// Brief: Master Arm Orientation Matching
FUNCTION_BLOCK PUBLIC FB_StateCtrlMatching EXTENDS FB_MasterArmCtrlBase
VAR_INPUT
END_VAR
VAR_OUTPUT
END_VAR
VAR
	// master-slave orientation match threshold
	m_matchAngleThres :LREAL := 2*g_deg2Rad;
	
	m_cmdRotInMonitor :Mat3d;
	
	m_initSolvedJntPos, m_iteSovlvedJntPos :Vec7d;
	m_IKSuccess :BOOL;
	
	m_matchTrajPlanner : FB_TrajMoveJ;
	m_targetJntPos :Vec7d;
	
	m_maxMatchJntVel:Vec7d:=[1.0, 1.0, 1.0, 2*pi, 3*pi, 3*pi, 5*pi];
	m_maxMatchJntAcc:Vec7d:=[1.0, 1.0, 1.0,  8*pi, 12*pi, 12*pi, 20*pi];
	m_maxMatchJntJerk:Vec7d:=[7(100.0)];
	
	m_rotErrAng :LREAL;

END_VAR

// override this function in each exact controller
METHOD PROTECTED calcCmdJntPos : BOOL

VAR_IN_OUT CONSTANT
	i_slaveIdx :INT;
	i_shoulderPose :ST_Frame;
	i_masterArm :FB_MasterArm;
	i_slaveStatus :ST_SlaveStatus;
END_VAR
var 
	i,j : INT;

	mq4,mq5,mq6,mq7:LREAL;
	q4,q5,q6,q7:LREAL;

	rotErr:Mat3d;
	wristRotInJnt3, wristRotInJnt4 :Mat3d;
	rot, invRot :Mat3d;
	cycleNum:INT;
	
	jnt4MoveRange:LREAL;
	jnt5Bias, jnt4MoveScale :LREAL;
	
	cmdJntErr:Vec7d;

END_VAR
IF m_IKSuccess THEN 
	// check if planner is ready
	IF  m_matchTrajPlanner.isGene = FALSE THEN
		RETURN;
	END_IF
	
	// traj plan
	calcCmdJntPos :=m_matchTrajPlanner.evaluate(m_timePeriod, jntPos=> m_cmdJntPos, jntVel=>m_cmdJntVel, jntAcc=> m_cmdJntAcc);
	
	vecSub(m_targetJntPos, m_cmdJntPos, cmdJntErr);
	
	matTranspose(i_masterArm.curCartPose.m_rot, invRot);
	matMultiply(invRot, m_cmdCartPose.m_rot, rotErr);
	rot2AngAxis(rotErr, angle=>m_rotErrAng,axis=>);
	m_isFinished := m_timePeriod > m_matchTrajPlanner.duration AND  norm(cmdJntErr)<g_jntCtrlAngTolHigh and abs(m_rotErrAng)<g_jntCtrlAngTolHigh;
	
	RETURN;
END_IF

// command rotation in monitor
m_cmdRotInMonitor := i_slaveStatus.m_curArmPose[i_slaveIdx].m_rot;

// command rotation in master arm base
matTranspose(i_shoulderPose.m_rot, invRot);
matMultiply(invRot, m_cmdRotInMonitor, m_cmdCartPose.m_rot);
m_cmdCartPose.m_pos:= i_masterArm.curCartPose.m_pos;

// calculate current orientation error
matTranspose(i_masterArm.curCartPose.m_rot, invRot);
matMultiply(invRot, m_cmdCartPose.m_rot, rotErr);
rot2AngAxis(rotErr, angle=>m_rotErrAng,axis=>);

// try IK with optimized posture
rot:=calcJnt3Rotation(m_cmdJntPos[1],m_cmdJntPos[2],m_cmdJntPos[3]);
matTranspose(rot, invRot);
matMultiply(invRot, m_cmdCartPose.m_rot, wristRotInJnt3);
IF 1=i_masterArm.armIdx THEN
	m_IKSuccess := leftWristOptIK(wristRotInJnt3,q4=>q4, q5=>q5, q6=>q6, q7=>q7);
ELSE
	m_IKSuccess := rightWristOptIK(wristRotInJnt3,q4=>q4, q5=>q5, q6=>q6, q7=>q7);
END_IF

// try IK with joint4 at minimal limit
IF NOT m_IKSuccess THEN
	q4:= GVL_ArmJointParameters.g_minJntPos[i_masterArm.armIdx,4];
	
	rot:=calcJnt4Rotation(m_cmdJntPos[1],m_cmdJntPos[2],m_cmdJntPos[3],q4);
	matTranspose(rot, invRot);
	matMultiply(invRot, m_cmdCartPose.m_rot, wristRotInJnt4);
	m_IKSuccess := wristIK(wristRotInJnt4,i_masterArm, q5=>q5, q6=>q6, q7=>q7);
END_IF

// try IK with joint4 at maximum limit
IF NOT m_IKSuccess THEN
	q4:= GVL_ArmJointParameters.g_maxJntPos[i_masterArm.armIdx,4];
	
	rot:=calcJnt4Rotation(m_cmdJntPos[1],m_cmdJntPos[2],m_cmdJntPos[3],q4);
	matTranspose(rot, invRot);
	matMultiply(invRot, m_cmdCartPose.m_rot, wristRotInJnt4);
	m_IKSuccess := wristIK(wristRotInJnt4,i_masterArm, q5=>q5, q6=>q6, q7=>q7);
END_IF

// minimize joint4 move angle
IF m_IKSuccess THEN
	
	// minimize based on join5 posture
	jnt4MoveRange :=  i_masterArm.jnt4LinkToMotor(m_targetJntPos[2],m_targetJntPos[3],q4)-i_masterArm.curJntPos[4];
	jnt5Bias :=  LIMIT (0, ABS(q5-pi), pi/2);
	jnt4MoveRange := jnt4MoveRange * ABS(COS(jnt5Bias));
	
	// minimize based on cartesian error
	IF ABS(m_rotErrAng)< 5.0 * g_deg2Rad THEN
		jnt4MoveRange := 0.0;
	END_IF
	
	mq4:=  i_masterArm.jnt4MotorToLink(m_targetJntPos[2],m_targetJntPos[3],i_masterArm.curJntPos[4] + jnt4MoveRange) ;
	
	rot:=calcJnt4Rotation(m_cmdJntPos[1],m_cmdJntPos[2],m_cmdJntPos[3],mq4);
	matTranspose(rot, invRot);
	matMultiply(invRot, m_cmdCartPose.m_rot, wristRotInJnt4);
	IF wristIK(wristRotInJnt4,i_masterArm, q5=>mq5, q6=>mq6, q7=>mq7) THEN
		q4:=mq4;
		q5:=mq5;
		q6:=mq6;
		q7:=mq7;
	END_IF
END_IF

// traj plan
IF m_IKSuccess THEN 
	m_targetJntPos:=m_cmdJntPos;
	m_targetJntPos[4]:=i_masterArm.jnt4LinkToMotor(m_targetJntPos[2],m_targetJntPos[3],q4);
	m_targetJntPos[5]:=q5;
	m_targetJntPos[6]:=q6;
	
	// roll flip handle
	i_masterArm.flipGripper(rollFlipHandle(i_masterArm.armIdx,i_masterArm.curJntPos[7], q7, o_cmdJntPos7 =>m_targetJntPos[7]));
	
	// no match for rotate joint if instrument is ultrasonic knife
	IF MasterArmControl.m_masterRobot.m_USKnifeRotClutch[i_slaveIdx] THEN
		m_targetJntPos[7] := i_masterArm.curJntPos[7];
	END_IF

	m_matchTrajPlanner.init(m_cmdJntPos,m_targetJntPos,m_maxMatchJntVel,m_maxMatchJntAcc,m_maxMatchJntJerk);
	m_timePeriod :=0;
END_IF
END_METHOD

// calculate joint3 rotation in arm coordinate
(*armDH=[   0      0   q1      d1;
            -deg90  0   q2      0;
            0       a3  q3      0];*)
METHOD PROTECTED calcJnt3Rotation : Mat3d
VAR_INPUT CONSTANT
	q1:LREAL;
	q2:LREAL;
	q3:LREAL;
END_VAR

VAR
	c1,c2,c3,s1,s2,s3,c23,s23 :LREAL;
END_VAR
// !Convert active joint position to DH model for kinematic calculation
q3:=q3-q2;  //q3=q8-q2

c1:=COS(q1);
c2:=COS(q2);
c3:=COS(q3);

s1:=SIN(q1);
s2:=SIN(q2);
s3:=SIN(q3);

c23:=COS(q2+q3);
s23:=SIN(q2+q3);

calcJnt3Rotation[1,1]:= c23*c1;
calcJnt3Rotation[2,1]:= c23*s1;
calcJnt3Rotation[3,1]:= -s23;

calcJnt3Rotation[1,2]:= -s23*c1;
calcJnt3Rotation[2,2]:= -s23*s1;
calcJnt3Rotation[3,2]:= -c23;

calcJnt3Rotation[1,3]:= -s1;
calcJnt3Rotation[2,3]:= c1;
calcJnt3Rotation[3,3]:=0;
END_METHOD

// calculate joint3 rotation in arm coordinate
(*[   0      0   q1      d1;
	-deg90  0   q2      0;
	0       a3  q3      0;
	 -deg90  a4  q4      d4]
*)
METHOD PROTECTED calcJnt4Rotation : Mat3d
VAR_INPUT
	q1 :LREAL;
	q2 :LREAL;
	q3 :LREAL;
	q4 :LREAL;// already at the link side
END_VAR

VAR
	c1,c2,c3,c4, s1,s2,s3,s4,c23,s23 :LREAL;
END_VAR
// !Convert active joint position to DH model for kinematic calculation
//q4:=q4+q3-q2-pi/2;//q4DH=q4motor+q8-q2-90;  
q3:=q3-q2;  //q3=q8-q2

c1:=COS(q1);
c2:=COS(q2);
c3:=COS(q3);
c4:=COS(q4);

s1:=SIN(q1);
s2:=SIN(q2);
s3:=SIN(q3);
s4:=SIN(q4);

c23:=COS(q2+q3);
s23:=SIN(q2+q3);

calcJnt4Rotation[1,1]:= s1*s4 + c4*c1*c23;
calcJnt4Rotation[2,1]:= - c1*s4 + c4*s1*c23;
calcJnt4Rotation[3,1]:= -s23*c4;

calcJnt4Rotation[1,2]:= c4*s1 - s4*c1*c23;
calcJnt4Rotation[2,2]:= -s4*s1*c23 - c1*c4;
calcJnt4Rotation[3,2]:=   s23*s4;

calcJnt4Rotation[1,3]:= -s23*c1;
calcJnt4Rotation[2,3]:= -s23*s1;
calcJnt4Rotation[3,3]:=-c23;
END_METHOD

PROPERTY IKSuccess : BOOL
GET
IKSuccess := m_IKSuccess;
END_GET
END_PROPERTY

METHOD PUBLIC init : BOOL
VAR_IN_OUT CONSTANT
	i_masterArm	:FB_MasterArm;
END_VAR
VAR_IN_OUT 
	r_masterArmCtrlCmd :ST_ArmCtrlCmds;
END_VAR
// check if to hold the command joint position unchanged
m_holdLastCmds := checkToHoldLastCmds(i_masterArm);

// init
SUPER^.Init(i_masterArm,r_masterArmCtrlCmd);

m_jntOPMode[4]:=DriverOPMode_PosTrq;
m_jntOPMode[5]:=DriverOPMode_PosTrq;
m_jntOPMode[6]:=DriverOPMode_PosTrq;
m_jntOPMode[7]:=DriverOPMode_PosTrq;

m_IKSuccess:=FALSE;
m_targetJntPos:=m_cmdJntPos;

// update commands to arm
copyCmds(r_masterArmCtrlCmd);
END_METHOD

// calculate command wrist joint position with an optimized posture
(*wristDH=[   -deg90  a4  q4      d4;
            deg90   0   q5      0;
            -deg90  0   q6      0;
            deg90   0   q7      0];*)
// set q6 = -pi/2 for desired posture
(* wristRot = 
[ COS(q7)*SIN(q4) - COS(q4)*SIN(q5)*SIN(q7), - SIN(q4)*SIN(q7) - COS(q4)*COS(q7)*SIN(q5), -COS(q4)*COS(q5)]
[                           cos(q5)*sin(q7),                             cos(q5)*cos(q7),         -sin(q5)]
[ cos(q4)*cos(q7) + sin(q4)*sin(q5)*sin(q7),   cos(q7)*sin(q4)*sin(q5) - cos(q4)*sin(q7),  cos(q5)*sin(q4)]
*)
METHOD PROTECTED leftWristOptIK : BOOL
VAR_IN_OUT CONSTANT
	i_cmdRot :Mat3d;
END_VAR
VAR_OUTPUT
	q4 :LREAL;
	q5 :LREAL;
	q6 :LREAL;
	q7 :LREAL;
END_VAR

VAR
	q51,q52 :LREAL;
	s4,c4,s5,c5,s7,c7:LREAL;
	q4UnreachPosMin: LREAL :=-pi/2;
	q4UnreachPosMax: LREAL :=45*g_deg2Rad;
	
END_VAR
q6:=-PI/2;
// q5 = [pi-135deg, pi+135deg]
q5 := ASIN(-i_cmdRot[2,3]);
q5:= PI-q5;

// q5=3pi/2 or q5=pi/2
IF ABS(q5-3*PI/2)<g_smallAng OR ABS(q5-PI/2)<g_smallAng THEN
	q4:= -pi;
	s7:= -i_cmdRot[1,1]/(COS(q4)*SIN(q5));
	c7:= i_cmdRot[3,1]/COS(q4);
	q7:=atan2(s7,c7);
	leftWristOptIK:=TRUE;
	RETURN;
END_IF

// solution one 
c5 :=COS(q5);
s7:=i_cmdRot[2,1]/c5;
c7:= i_cmdRot[2,2]/c5;
q7:=atan2(s7,c7);

//q4=[-pi/2-225deg, -pi/2]
c4 := -i_cmdRot[1,3]/c5;
s4:= i_cmdRot[3,3]/c5;
q4:=atan2(s4,c4);
IF q4> GVL_ArmJointParameters.g_minJntPos[1,4] AND q4<GVL_ArmJointParameters.g_maxJntPos[1,4] THEN
	leftWristOptIK:=TRUE;
	RETURN;
ELSIF q4> GVL_ArmJointParameters.g_maxJntPos[1,4] AND q4-2*pi> GVL_ArmJointParameters.g_minJntPos[1,4] THEN
	q4:=q4-2*PI;
	leftWristOptIK:=TRUE;
	RETURN;
END_IF

// solution2
IF q5 > pi THEN
	q5 := 3*PI-q5;
ELSE
	q5:= pi-q5;
END_IF
IF q5 > GVL_ArmJointParameters.g_maxJntPos[1,5] OR q5<GVL_ArmJointParameters.g_minJntPos[1,5] THEN
	leftWristOptIK:=FALSE;
	RETURN;
END_IF

c5 :=COS(q5);
s7:=i_cmdRot[2,1]/c5;
c7:= i_cmdRot[2,2]/c5;
q7:=atan2(s7,c7);

c4 := -i_cmdRot[1,3]/c5;
s4:= i_cmdRot[3,3]/c5;
q4:=atan2(s4,c4);
IF q4> GVL_ArmJointParameters.g_minJntPos[1,4] AND q4<GVL_ArmJointParameters.g_maxJntPos[1,4] THEN
	leftWristOptIK:=TRUE;
	RETURN;
ELSIF q4> GVL_ArmJointParameters.g_maxJntPos[1,4] AND q4-2*pi< GVL_ArmJointParameters.g_minJntPos[1,4] THEN
	q4:=q4-2*PI;
	leftWristOptIK:=TRUE;
	RETURN;
END_IF
END_METHOD

// calculate command wrist joint position with an optimized posture
(*wristDH=[   -deg90  a4  q4      d4;
            deg90   0   q5      0;
            -deg90  0   q6      0;
            deg90   0   q7      0];*)
// set q6 = pi/2 for desired posture
(* wristRot = 
[ - cos(q7)*sin(q4) - cos(q4)*sin(q5)*sin(q7), sin(q4)*sin(q7) - cos(q4)*cos(q7)*sin(q5),  cos(q4)*cos(q5)]
[                             cos(q5)*sin(q7),                           cos(q5)*cos(q7),          sin(q5)]
[   sin(q4)*sin(q5)*sin(q7) - cos(q4)*cos(q7), cos(q4)*sin(q7) + cos(q7)*sin(q4)*sin(q5), -cos(q5)*sin(q4)]
 
*)
METHOD PROTECTED rightWristOptIK : BOOL
VAR_IN_OUT CONSTANT
	i_cmdRot :Mat3d;
END_VAR
VAR_OUTPUT
	q4 :LREAL;
	q5 :LREAL;
	q6 :LREAL;
	q7 :LREAL;
END_VAR

VAR
	q51,q52 :LREAL;
	s4,c4,s5,c5,s7,c7:LREAL;
	q4UnreachPosMin: LREAL :=-pi/2;
	q4UnreachPosMax: LREAL :=45*g_deg2Rad;
	
END_VAR
q6:=PI/2;
// q5 = [pi-135deg, pi+135deg]
q5 := ASIN(i_cmdRot[2,3]);
q5:= PI-q5;

// q5=3pi/2 or q5=pi/2
IF ABS(q5-3*PI/2)<g_smallAng OR ABS(q5-PI/2)<g_smallAng THEN
	q4:= 0;
	s7:= -i_cmdRot[1,1]/(COS(q4)*SIN(q5));
	c7:= -i_cmdRot[3,1]/COS(q4);
	q7:=atan2(s7,c7);
	rightWristOptIK:=TRUE;
	RETURN;
END_IF

// solution one 
c5 :=COS(q5);
s7:=i_cmdRot[2,1]/c5;
c7:= i_cmdRot[2,2]/c5;
q7:=atan2(s7,c7);

//q4=[-pi/2, -pi/2+225deg]
c4 := i_cmdRot[1,3]/c5;
s4:= -i_cmdRot[3,3]/c5;
q4:=atan2(s4,c4);
IF q4> GVL_ArmJointParameters.g_minJntPos[2,4] AND q4<GVL_ArmJointParameters.g_maxJntPos[2,4] THEN
	rightWristOptIK:=TRUE;
	RETURN;
END_IF

// solution2
IF q5 > pi THEN
	q5 := 3*PI-q5;
ELSE
	q5:= pi-q5;
END_IF
IF q5 > GVL_ArmJointParameters.g_maxJntPos[1,5] OR q5<GVL_ArmJointParameters.g_minJntPos[1,5] THEN
	rightWristOptIK:=FALSE;
	RETURN;
END_IF

c5 :=COS(q5);
s7:=i_cmdRot[2,1]/c5;
c7:= i_cmdRot[2,2]/c5;
q7:=atan2(s7,c7);

//q4=[-pi/2, -pi/2+225deg]
c4 := i_cmdRot[1,3]/c5;
s4:= -i_cmdRot[3,3]/c5;
q4:=atan2(s4,c4);
IF q4> GVL_ArmJointParameters.g_minJntPos[2,4] AND q4<GVL_ArmJointParameters.g_maxJntPos[2,4] THEN
	rightWristOptIK:=TRUE;
	RETURN;
END_IF
END_METHOD

METHOD PROTECTED rollFlipHandle : BOOL
VAR_INPUT
	i_armIdx:INT;
	i_curJntPos7 :LREAL;
	i_initCmdJntPos7 :LREAL;
END_VAR
VAR_OUTPUT
	o_cmdJntPos7 :LREAL;
END_VAR

VAR
	solFeasible1,solFeasible2 :BOOL;
	solIdx :INT:=0;
	halfcycleNum1, halfcycleNum2:INT;
	solution1, solution2 :LREAL;
END_VAR
// this part is used to drive gripper back near center, in case that gripper roll is stuck near limit
// TODO: remove after gripper roll has infinite motion range
IF NOT (MasterArmControl.m_masterInputDataPool.m_cartStatus.m_surgonReady) THEN
	o_cmdJntPos7:=i_initCmdJntPos7;
	rollFlipHandle:=FALSE;
	RETURN;
END_IF

// handle multiple cycles of joint7
// find the first solution within pi from current position
halfcycleNum1 := LREAL_TO_INT((i_curJntPos7 - i_initCmdJntPos7)/pi);
solution1 := halfcycleNum1 * pi + i_initCmdJntPos7;

// solution2
IF solution1 > i_curJntPos7 THEN
	solution2 := solution1 - PI;
	halfcycleNum2 := halfcycleNum1 - 1;
ELSE
	solution2 := solution1 + PI;
	halfcycleNum2 := halfcycleNum1 + 1;
END_IF

//choose the solution which is closer to current q7 which can achive orientation match with a max pi/2 degree
// NOTE: There maybe risk this joint7 is stuck at limit, which can be solved after joint7 has infinite rotation angle,
solFeasible1:=solution1> GVL_ArmJointParameters.g_minJntPos[i_armIdx,7] AND solution1< GVL_ArmJointParameters.g_maxJntPos[i_armIdx,7];
solFeasible2:=solution2> GVL_ArmJointParameters.g_minJntPos[i_armIdx,7] AND solution2< GVL_ArmJointParameters.g_maxJntPos[i_armIdx,7];
IF solFeasible1 AND solFeasible2 THEN
	IF ABS(solution1-i_curJntPos7) < ABS(solution2-i_curJntPos7)  THEN
		solIdx:=1;
	ELSE
		solIdx:=2;
	END_IF
ELSIF solFeasible1 AND NOT(solFeasible2) THEN
	solIdx:=1;
ELSIF solFeasible2 AND NOT(solFeasible1) THEN
	solIdx:=2;
ELSE
	solIdx:=0;
END_IF

IF solIdx = 1 THEN
	o_cmdJntPos7 := solution1;
	rollFlipHandle:= ((ABS(halfcycleNum1) MOD 2) = 1);
ELSIF solIdx =2 THEN
	o_cmdJntPos7 := solution2;
	rollFlipHandle:= ((ABS(halfcycleNum2) MOD 2) = 1);
ELSE
	o_cmdJntPos7:=i_initCmdJntPos7;
	rollFlipHandle:=FALSE;
END_IF
END_METHOD

// calculate position of joint 5/6/7 
(*wristDH=[   deg90   0   q5      0;
            -deg90  0   q6      0;
            deg90   0   q7      0];*)
(* wristRot = 
[ cos(q5)*cos(q6)*cos(q7) - sin(q5)*sin(q7), - cos(q7)*sin(q5) - cos(q5)*cos(q6)*sin(q7), cos(q5)*sin(q6)]
[                           cos(q7)*sin(q6),                            -sin(q6)*sin(q7),        -cos(q6)]
[ cos(q5)*sin(q7) + cos(q6)*cos(q7)*sin(q5),   cos(q5)*cos(q7) - cos(q6)*sin(q5)*sin(q7), sin(q5)*sin(q6)]
*)
METHOD PROTECTED wristIK : BOOL
VAR_IN_OUT CONSTANT
	i_cmdRot :Mat3d;
	i_masterArm :FB_MasterArm;
END_VAR

VAR_OUTPUT
	q5:	LREAL;
	q6:	LREAL;
	q7:	LREAL;
END_VAR

VAR
	invRot :Mat3d;
	jnt4Rotation :Mat3d;
	s5, s7, c5, c7:LREAL;
END_VAR
// calculate wrist joint position
// q6=[-pi/2-45deg, -pi/2+45deg]
IF 1 = i_masterArm.armIdx THEN
	q6:= -ACOS(-i_cmdRot[2,3]);
// q6=[pi/2-45deg, pi/2+45deg]
ELSE
	q6:= ACOS(-i_cmdRot[2,3]);
END_IF

IF q6>GVL_ArmJointParameters.g_maxJntPos[i_masterArm.armIdx, 6] OR q6< GVL_ArmJointParameters.g_minJntPos[i_masterArm.armIdx, 6] THEN
	wristIK:=FALSE;
	RETURN;
END_IF

// q5 = [pi-135deg, pi+135deg]
c5 := i_cmdRot[1,3]/SIN(q6);
s5 := i_cmdRot[3,3]/SIN(q6);
q5:=atan2(s5,c5);
IF q5<GVL_ArmJointParameters.g_minJntPos[1,5] THEN
	q5:=q5+2*PI;
END_IF
IF q5>GVL_ArmJointParameters.g_maxJntPos[1,5]THEN
	wristIK:=FALSE;
	RETURN;
END_IF
c7 := i_cmdRot[2,1]/SIN(q6);
s7 := -i_cmdRot[2,2]/SIN(q6);
q7:=atan2(s7,c7);
wristIK:=true;
END_METHOD

END_FUNCTION_BLOCK

(* stored: Version 1.1.0.1, ProductVersion 3.1.4024.12
   POU FB_StateCtrlMatching: Id {886a3c3b-c6fb-4a12-8c63-bddb11202d66}, SpecialFunc None
   Method calcCmdJntPos: Id {51b8574c-dbe7-40e3-8c59-ca4f0064a75b}
   Method calcJnt3Rotation: Id {45e74725-458c-4f96-a988-7b138ad9e9c4}
   Method calcJnt4Rotation: Id {7c3dafce-1980-4f86-996d-7fbd85661296}
   Property IKSuccess: Id {472fdaf7-37fe-4950-9971-249f506f982b}
   Get Get: Id {ee890eed-eea0-42af-913f-a01a7cf1da04}
   Method init: Id {af3225b4-51f5-49e0-8b94-24f1ab0678fd}
   Method leftWristOptIK: Id {0caeaf17-79dd-44c1-86e3-89513a734de0}
   Method rightWristOptIK: Id {b0cf9587-0a5e-4160-99d0-26fa71dc5b57}
   Method rollFlipHandle: Id {8ed883c8-bcc7-4a8d-b5a5-e09032451118}
   Method wristIK: Id {5d6388c7-a5fc-4ec4-bbd8-54b7da79fe62} *)
